Staubli VAL3: HRAS_trial.pjx

--- HRAS_trial.pjx ---
Parameters version=s7.10.2 stackSize=5000 millimeterUnit=true
Program file=calculate_pick.pgx
Program file=calculate_rc.pgx
Program file=calculate_total.pgx
Program file=check_out_set.pgx
Program file=f2_place.pgx
Program file=pick_cells.pgx
Program file=pp_auto_v1.pgx
Program file=pp_auto_v2.pgx
Program file=pp_bs_f1f2f3.pgx
Program file=pp_bs_f2f3.pgx
Program file=pp_cell_bk_f123.pgx
Program file=pp_cell_bk_f2f3.pgx
Program file=pp_cells.pgx
Program file=pp_shelf.pgx
Program file=regular_pick.pgx
Program file=regular_place.pgx
Program file=return_config.pgx
Program file=show_check.pgx
Program file=show_menu.pgx
Program file=show_progress.pgx
Program file=start.pgx
Program file=stop.pgx
Data file=HRAS_trial.dtx
Type name=vacuumSet path=Disk://designr0/designr0.pjx

--- HRAS_trial.dtx ---
dio dDio_t1_vb = {link=BasicIO-1\%Q1}
dio dDio_t1_vg
dio dDio_t1_vs = {link=fIn0}
dio dDio_t3_vb
dio dDio_t3_vg
dio dDio_t3_vs = {link=fIn0}
frame f1 = {x=-139.3, y=417.51507, z=-171.375326, rz=179.999983, fatherId=world[0]}
frame f2 = {x=-0.751213, y=410.035294, z=-169.439088, rz=179.999983, fatherId=world[0]}
frame f3 = {x=-105.214041, y=542.677355, z=-169.567493, rz=-89.997724, fatherId=world[0]}
frame fixture = {x=-479.290297, y=224.508367, z=-148, rz=-90.00005, fatherId=world[0]}
frame shelf = {x=-472.219676, y=345.637635, z=-165, rz=-90, fatherId=world[0]}
mdesc mNomSpeed
mdesc mSlowSpeed = {accel=50, vel=10, decel=50}
num nNum_blow_delay = 1
num nNum_blow_h = 0.5
num nNum_press = 4
num nNum_safe_h = 50
pointRx f1pick = {x=43.79, y=-7, z=0.5, rx=-180, rz=-180, fatherId=shelf[0]}
pointRx f1picksafe = {x=43.79, y=-7, z=20, rx=180, rz=-180, fatherId=shelf[0]}
pointRx f1place = {x=20, y=-19.98, rx=-180, rz=-180, fatherId=fixture[0]}
pointRx f1placesafe = {x=20, y=-19.98, z=20, rx=-180, rz=180, fatherId=fixture[0]}
pointRx f2pick = {x=29.79, y=-6.4, z=0.5, rx=-180, rz=180, fatherId=shelf[0]}
pointRx f2picksafe = {x=29.79, y=-6.4, z=20, rx=-180, rz=179, fatherId=shelf[0]}
pointRx f2place = {x=20, y=-16.82, rx=-180, rz=-180, fatherId=fixture[0]}
pointRx f2placesafe = {x=20, y=-16.82, z=20, rx=-180, rz=180, fatherId=fixture[0]}
pointRx f3pick = {x=7.79, y=-6.75, z=0.5, rx=-180, wrist=wpositive, fatherId=shelf[0]}
pointRx f3picksafe = {x=7.790741, y=-6.500263, z=50, rx=-179.999806, ry=-0.000248, rz=-2.000096, fatherId=shelf[0]}
pointRx f3place = {x=20, y=-16.62, z=3.8, rx=180, fatherId=fixture[0]}
pointRx f3placesafe = {x=20.000011, y=-16.619972, z=20, rx=-179.999664, ry=0.000116, rz=3E-06, fatherId=fixture[0]}
pointRx origin = {rx=-180, rz=-180, fatherId=fixture[0]}
pointRx pPointRx_f1_lb = {x=8.1, y=23.5, z=1.8, rx=180, fatherId=f1[0]}
pointRx pPointRx_f2_lb = {x=-3.5, y=25, z=0.2, rx=180, fatherId=f2[0]}
pointRx pPointRx_f3_lb = {x=28.5, y=3.34, z=0.2, rx=-180, rz=-180, fatherId=f3[0]}
pointRx ref = {x=-188.838954, y=475.816737, z=-162.486188, rx=180, rz=180, fatherId=world[0]}
screen sScreen_menu
screen sScreen_ppShelf
tool ca = {z=55, rz=45, fatherId=flange[0], ioLink=valve1}
tool t1 = {y=-18.5, fatherId=ca[0], ioLink=BasicIO-1\%Q0, ioOpen=1, ioClose=0.5}
tool t2 = {y=-4.5, fatherId=ca[0], ioLink=valve1}
tool t3 = {y=17.5, fatherId=ca[0], ioLink=BasicIO-1\%Q2, ioOpen=0.5, ioClose=0.5}
dio dDio_t1_cy
dio dDio_t2_cy
dio dDio_t3_cy

--- start.pgx ---
program start()
  local num l_nNum_choosen
begin
  resetMotion()

  //----------------------
  //  Reset I/O
  //----------------------
  call check_out_set(t1.gripper,false)
  call check_out_set(t2.gripper,false)
  call check_out_set(t3.gripper,false)

  call check_out_set(dDio_f1_fit,false)
  call check_out_set(dDio_bk,false)

  call check_out_set(dDio_f1_secure,false)
  call check_out_set(dDio_f2_secure,false)
  call check_out_set(dDio_f3_secure,false)

  call check_out_set(dDio_t1_cy,false)
  call check_out_set(dDio_t2_cy,false)
  call check_out_set(dDio_t3_cy,false)
  //----------------------
  //  Reset I/O
  //----------------------

  call show_menu(sScreen_ppShelf,l_nNum_choosen)

  while true
    switch l_nNum_choosen
      case 271
        //F1
        call pick_cells(1)
      break
      case 272
        //F2
        call pick_cells(2)
      break
      case 273
        //F3
        call pick_cells(3)
      break
      case 274
        //F4
        call pp_shelf()
      break
      case 275
        //F5
        call pp_cells()
      break
      //----------------------
      //
      //----------------------
      case 276
        //F6
        call pp_bs_f2f3()
      break
      case 277
        //F7
        call pp_auto_v1()
      break
      case 278
        //F8
        call pp_auto_v2()
      break
      case 113
        //q
        call pp_bs_f1f2f3()
      break
      default
        return
      break
    endSwitch
  endWhile

end

--- calculate_pick.pgx ---
public program calculate_pick(num x_nNum_row, num x_nNum_col, point& x_pPoint_return, num x_nNum_choose)
  local num l_nNum_pitchX
  local num l_nNum_pitchY
  local point l_pPoint_lb
begin
  //given row,col(z-based, count from left-bottom)
  //return position


  //set left-bottom corner position and pitch
  switch x_nNum_choose
    case 1
      //f1
      l_nNum_pitchX = 6.6
      l_nNum_pitchY = 11.3

      l_pPoint_lb = pPointRx_f1_lb
    break
    case 2
      //f2
      l_nNum_pitchX = 8
      l_nNum_pitchY = 10

      l_pPoint_lb = pPointRx_f2_lb
    break
    case 3
      //f3
      l_nNum_pitchX = -14
      l_nNum_pitchY = 22

      l_pPoint_lb = pPointRx_f3_lb
    break
    case 4
      //bottom
      l_nNum_pitchX = 32
      l_nNum_pitchY = 33

      l_pPoint_lb = pPointRx_bt_lb
    break

  endSwitch


  x_pPoint_return = l_pPoint_lb

  x_pPoint_return.trsf.x = x_pPoint_return.trsf.x + x_nNum_col * l_nNum_pitchX
  x_pPoint_return.trsf.y = x_pPoint_return.trsf.y + x_nNum_row * l_nNum_pitchY

  //---------------------------------------------
  // Bottom part special case - base frame offset
  //---------------------------------------------
  switch x_nNum_choose
    case 4
      fFrame_ofs.trsf.x = x_nNum_col * l_nNum_pitchX
      fFrame_ofs.trsf.y = x_nNum_row * l_nNum_pitchY
      //maintain the lb point
      x_pPoint_return = pPointRx_bt_lb
    break
  endSwitch

end

--- calculate_rc.pgx ---
program calculate_rc(num x_nNum_index, num x_nNum_choose, num& x_nNum_cRow, num& x_nNum_cCol)
  local num l_nNum_lCol
  local num l_nNum_lRow
begin

  call return_config(x_nNum_choose,l_nNum_lRow,l_nNum_lCol)

  //Quotien
  x_nNum_cRow = roundDown(x_nNum_index / (l_nNum_lCol + 1))
  //Modulo reminder
  x_nNum_cCol = x_nNum_index % (l_nNum_lCol+1)


end

--- calculate_total.pgx ---
program calculate_total(num x_nNum_choose, num& x_nNum_total)
  local num l_nNum_lCol
  local num l_nNum_lRow
begin
  call return_config(x_nNum_choose,l_nNum_lRow,l_nNum_lCol)
    //(max index)
  x_nNum_total = (l_nNum_lRow + 1) * (l_nNum_lCol+1)
end

--- check_out_set.pgx ---
program check_out_set(dio x_dDio_target, bool x_bBool_onoff)
begin
  if ioStatus(x_dDio_target) >= 0
    //once io is working
    x_dDio_target = x_bBool_onoff
  endIf
end

--- f1_cell_count.pgx ---
program f1_cell_count()
begin
  //given row,col , return position
  //retunr position
end

--- f1_cell_pick.pgx ---
program f1_cell_pick()
begin
  //pick from f1 put to bin
end

--- f2_place.pgx ---
program f2_place(mdesc x_mMdesc, mdesc x_mMdesc_slow)
  local point l_pPoint_blow
  local point l_pPoint_drop
  local point l_pPoint_safe
begin
  //vertical drop filter-2 process

  //control point preparation
  l_pPoint_safe=f2place
  l_pPoint_safe.trsf.z=l_pPoint_safe.trsf.z+nNum_safe_h

  l_pPoint_blow=f2place
  l_pPoint_blow.trsf.z=l_pPoint_blow.trsf.z+nNum_blow_h

  l_pPoint_drop=f2place

  ////to place via safe
  movej(l_pPoint_safe,t1,x_mMdesc)
  movej(l_pPoint_drop,t1,x_mMdesc)
  waitEndMove()
  //vg off
  if ioStatus(t1.gripper) >= 0
    close(t1)
  endIf
  if ioStatus(dDio_t1_vb) >= 0
    dDio_t1_vb=true
  endIf

    //on and delay
    delay(nNum_blow_delay)
    //to blow end
    movej(l_pPoint_blow,t1,x_mMdesc_slow)
    waitEndMove()
  //vb off
  if ioStatus(dDio_t1_vb) >= 0
     dDio_t1_vb=false
  endIf

    //to safe
    movej(l_pPoint_safe,t1,x_mMdesc)
    waitEndMove()
end

--- key_check.pgx ---
program key_check(string x_sString_show (dimensions=1))
begin
  userPage(sScreen_ppShelf)
  title(sScreen_ppShelf,x_sString_show)
  gotoxy(sScreen_ppShelf,0,6)
  putln(sScreen_ppShelf,"Press any key")
  //anykey
  get(sScreen_ppShelf)
  cls(sScreen_ppShelf)
end

--- pick_cells.pgx ---
program pick_cells(num x_nNum_choose)
  local num l_nNum_cRow
  local num l_nNum_cCol
  local point l_pPoint_cur
  local tool l_tTool_cur
  local point l_pPoint_lb_cur
  local num l_nNum_total
  local num l_nNum_current
  local dio l_dDio_cur_cy
  local dio l_dDio_secure
begin
  //pick from f1 put to bin
  call show_check("Reload")

  switch x_nNum_choose
    case 1
      //f1
      l_tTool_cur = t1
      dioLink(l_dDio_cur_cy,dDio_t1_cy)
      dioLink(l_dDio_secure,dDio_f1_secure)
      //dio assignment
    break
    case 2
      //f2
      l_tTool_cur = t2
      dioLink(l_dDio_cur_cy,dDio_t2_cy)
      dioLink(l_dDio_secure,dDio_f2_secure)
      //dio assignment
    break
    case 3
      //f3
      l_tTool_cur = t3
      dioLink(l_dDio_cur_cy,dDio_t3_cy)
      dioLink(l_dDio_secure,dDio_f3_secure)
      //dio assignment
    break

  endSwitch

  //calculate total
  call calculate_total(x_nNum_choose,l_nNum_total)

  for l_nNum_current=0 to(l_nNum_total-1) step 1

    //show progress
    call show_progress(sScreen_ppShelf,l_nNum_current+1,l_nNum_total,6)

    //row,col count
    call calculate_rc(l_nNum_current,x_nNum_choose,l_nNum_cRow,l_nNum_cCol)
    //pick position count
    call calculate_pick(l_nNum_cRow,l_nNum_cCol,l_pPoint_cur,x_nNum_choose)
    //pick (not defined yet
    call regular_pick(l_tTool_cur,mNomSpeed,mSlowSpeed,l_pPoint_cur,l_dDio_cur_cy,false,l_dDio_secure)

    //bin place (bin not defined yet
    call regular_place(l_tTool_cur,mNomSpeed,mSlowSpeed,ref,false,l_dDio_cur_cy,false)

  endFor

end

--- pickNplaceShelf.pgx ---
program pickNplaceShelf()
begin
  //assumption : arm in cal_ref1

  //pick f1
  //wait until user confirm (reload bottom
  //place f1
  //pick f2
  //wait until user confirm (close the fixture
  //place f2 (need blow simultanously
  //pick f3
  //place f3

end

--- place_f2.pgx ---
program place_f2()
begin
  //safe height
  //place
  //shut off
  dDio_t1_vg = off
  //back with blow

end

--- pp_auto_v1.pgx ---
program pp_auto_v1()
  local num l_nNum_bt_lim
  local num l_nNum_bt_idx
  local num l_nNum_f3_idx
  local num l_nNum_f2_idx
  local num l_nNum_f1_idx
  local num l_nNum_f3_lim
  local num l_nNum_f2_lim
  local num l_nNum_f1_lim
  local num l_nNum_cRow
  local num l_nNum_cCol
  local point l_pPoint_cur
begin
  //-----------------------------------------
  //  Cells to manual fixture
  //-----------------------------------------

  //initialize
  call calculate_total(1,l_nNum_f1_lim)
  call calculate_total(2,l_nNum_f2_lim)
  call calculate_total(3,l_nNum_f3_lim)
  call calculate_total(4,l_nNum_bt_lim)

  l_nNum_f1_idx = 0
  l_nNum_f2_idx = 0
  l_nNum_f3_idx = 0
  l_nNum_bt_idx = 0

  while true

    call show_check("Unload ASSY. filter")

    //------------
    //bottom cell pick
    //------------
    //runout remider
    if l_nNum_bt_idx >= l_nNum_bt_lim
      //warning if runs out
      call show_check("Reload Bottom")
      //reset
      l_nNum_bt_idx = 0
    endIf


    call calculate_rc(l_nNum_bt_idx,4,l_nNum_cRow,l_nNum_cCol)
    call calculate_pick(l_nNum_cRow,l_nNum_cCol,l_pPoint_cur,4)
    call regular_pick(t3,mNomSpeed,mSlowSpeed,l_pPoint_cur,dDio_t3_cy,false,dDio_f3_secure)

    //show progress
    call show_progress(sScreen_ppShelf,l_nNum_bt_idx+1,l_nNum_bt_lim,5)
    //increase
    l_nNum_bt_idx = l_nNum_bt_idx +1

    //------------
    //bottom place
    //------------
    call regular_place(t3,mNomSpeed,mSlowSpeed,pPointRx_bt_pos,false,dDio_t3_cy,false)

    //------------
    //f1 cell pick
    //------------

    //runout remider
    if l_nNum_f1_idx >= l_nNum_f1_lim
      //warning if runs out
      call show_check("Reload F1")
      //reset
      l_nNum_f1_idx = 0
    endIf

    call calculate_rc(l_nNum_f1_idx,1,l_nNum_cRow,l_nNum_cCol)
    call calculate_pick(l_nNum_cRow,l_nNum_cCol,l_pPoint_cur,1)
    call regular_pick(t1,mNomSpeed,mSlowSpeed,l_pPoint_cur,dDio_t1_cy,false,dDio_f1_secure)

    //show progress
    call show_progress(sScreen_ppShelf,l_nNum_f1_idx+1,l_nNum_f1_lim,6)
    //increase
    l_nNum_f1_idx = l_nNum_f1_idx +1

    //----------
    //f2 cell pick
    //------------

    //runout remider
    if l_nNum_f2_idx >= l_nNum_f2_lim
      //warning if runs out
      call show_check("Reload F2")
      //reset
      l_nNum_f2_idx = 0
    endIf


    call calculate_rc(l_nNum_f2_idx,2,l_nNum_cRow,l_nNum_cCol)
    call calculate_pick(l_nNum_cRow,l_nNum_cCol,l_pPoint_cur,2)
    call regular_pick(t2,mNomSpeed,mSlowSpeed,l_pPoint_cur,dDio_t2_cy,false,dDio_f2_secure)
    //show progress
    call show_progress(sScreen_ppShelf,l_nNum_f2_idx+1,l_nNum_f2_lim,7)
    //increase
    l_nNum_f2_idx = l_nNum_f2_idx +1

    //-------
    //f3pick
    //-------

    //runout reminder
    if l_nNum_f3_idx >= l_nNum_f3_lim
      //warning if runs out
      call show_check("Reload F3")
      //reset
      l_nNum_f3_idx = 0
    endIf
    call calculate_rc(l_nNum_f3_idx,3,l_nNum_cRow,l_nNum_cCol)
    call calculate_pick(l_nNum_cRow,l_nNum_cCol,l_pPoint_cur,3)
    call regular_pick(t3,mNomSpeed,mSlowSpeed,l_pPoint_cur,dDio_t3_cy,false,dDio_f3_secure)

    //show progress
    call show_progress(sScreen_ppShelf,l_nNum_f3_idx+1,l_nNum_f3_lim,8)
    //increase
    l_nNum_f3_idx = l_nNum_f3_idx +1

    //-------------
    // Back secure
    //-------------
    call pp_bs_f2f3()

    //----------------
    // F1, F2+F3 place
    //----------------
    call regular_place(t1,mNomSpeed,mSlowSpeed,pPointRx_f1_pos,false,dDio_t1_cy,false)
    // put  f1 fit
    if ioStatus(dDio_f1_fit) >= 0
      dDio_f1_fit = true
      delay(nNum_cy_delay)
    endIf
    //f3place
    call regular_place(t3,mNomSpeed,mSlowSpeed,pPointRx_f3_pos,false,dDio_t3_cy,false)
    // off  f1 fit
    if ioStatus(dDio_f1_fit) >= 0
      dDio_f1_fit = false
    endIf

  endWhile


end

--- pp_auto_v2.pgx ---
program pp_auto_v2(bool x_bBool_single)
  local num l_nNum_bt_lim
  local num l_nNum_bt_idx
  local num l_nNum_f3_idx
  local num l_nNum_f2_idx
  local num l_nNum_f1_idx
  local num l_nNum_f3_lim
  local num l_nNum_f2_lim
  local num l_nNum_f1_lim
  local num l_nNum_cRow
  local num l_nNum_cCol
  local point l_pPoint_cur
begin
  //-----------------------------------------
  //  Cells to manual fixture
  //-----------------------------------------

  //initialize
  call calculate_total(1,l_nNum_f1_lim)
  call calculate_total(2,l_nNum_f2_lim)
  call calculate_total(3,l_nNum_f3_lim)
  call calculate_total(4,l_nNum_bt_lim)

  l_nNum_f1_idx = 0
  l_nNum_f2_idx = 0
  l_nNum_f3_idx = 0
  l_nNum_bt_idx = 0

  while true

    call show_check("Unload ASSY. filter")

    if x_bBool_single == true
      //prompt reminder
      l_nNum_bt_idx = l_nNum_bt_lim
    endIf

    //------------
    //bottom cell pick
    //------------
    //runout remider
    if l_nNum_bt_idx >= l_nNum_bt_lim
      //warning if runs out
      call show_check("Reload Bottom")
      //reset
      l_nNum_bt_idx = 0
    endIf

    call calculate_rc(l_nNum_bt_idx,4,l_nNum_cRow,l_nNum_cCol)
    call calculate_pick(l_nNum_cRow,l_nNum_cCol,l_pPoint_cur,4)
    call regular_pick(t3,mNomSpeed,mSlowSpeed,l_pPoint_cur,dDio_t3_cy,false,dDio_f3_secure)


    //show progress
    call show_progress(sScreen_ppShelf,l_nNum_bt_idx+1,l_nNum_bt_lim,5)
    //increase
    l_nNum_bt_idx = l_nNum_bt_idx +1

    //------------
    //bottom place
    //------------
    call regular_place(t3,mNomSpeed,mSlowSpeed,pPointRx_bt_pos,false,dDio_t3_cy,false)

    //------------
    //f1 cell pick
    //------------

    //runout remider
    if l_nNum_f1_idx >= l_nNum_f1_lim
      //warning if runs out
      call show_check("Reload F1")
      //reset
      l_nNum_f1_idx = 0
    endIf

    call calculate_rc(l_nNum_f1_idx,1,l_nNum_cRow,l_nNum_cCol)
    call calculate_pick(l_nNum_cRow,l_nNum_cCol,l_pPoint_cur,1)
    call regular_pick(t1,mNomSpeed,mSlowSpeed,l_pPoint_cur,dDio_t1_cy,false,dDio_f1_secure)

    //show progress
    call show_progress(sScreen_ppShelf,l_nNum_f1_idx+1,l_nNum_f1_lim,6)
    //increase
    l_nNum_f1_idx = l_nNum_f1_idx +1

    //----------
    //f2 cell pick
    //------------

    //runout remider
    if l_nNum_f2_idx >= l_nNum_f2_lim
      //warning if runs out
      call show_check("Reload F2")
      //reset
      l_nNum_f2_idx = 0
    endIf


    call calculate_rc(l_nNum_f2_idx,2,l_nNum_cRow,l_nNum_cCol)
    call calculate_pick(l_nNum_cRow,l_nNum_cCol,l_pPoint_cur,2)
    call regular_pick(t2,mNomSpeed,mSlowSpeed,l_pPoint_cur,dDio_t2_cy,false,dDio_f2_secure)
    //show progress
    call show_progress(sScreen_ppShelf,l_nNum_f2_idx+1,l_nNum_f2_lim,7)
    //increase
    l_nNum_f2_idx = l_nNum_f2_idx +1

    //-------
    //f3pick
    //-------

    //runout reminder
    if l_nNum_f3_idx >= l_nNum_f3_lim
      //warning if runs out
      call show_check("Reload F3")
      //reset
      l_nNum_f3_idx = 0
    endIf
    call calculate_rc(l_nNum_f3_idx,3,l_nNum_cRow,l_nNum_cCol)
    call calculate_pick(l_nNum_cRow,l_nNum_cCol,l_pPoint_cur,3)
    call regular_pick(t3,mNomSpeed,mSlowSpeed,l_pPoint_cur,dDio_t3_cy,false,dDio_f3_secure)

    //show progress
    call show_progress(sScreen_ppShelf,l_nNum_f3_idx+1,l_nNum_f3_lim,8)
    //increase
    l_nNum_f3_idx = l_nNum_f3_idx +1

    //-------------
    // Back secure (F1,F2,F3
    //-------------
    call pp_bs_f1f2f3()
    //-------------
    // F1,F2,F3 pick at once
    //-------------
    call regular_pick(t3,mNomSpeed,mSlowSpeed,pPointRx_f3_bk,dDio_t3_cy,false,dDio_f3_secure)
    //----------------
    // F1+F2+F3 place at once
    //----------------
    //f3place
    call regular_place(t3,mNomSpeed,mSlowSpeed,pPointRx_f3_pos,false,dDio_t3_cy,false)

  endWhile


end

--- pp_back_secure.pgx ---
program pp_back_secure()
begin
  //given f2,f3 are in hand
  //exit state : f2, f3 secured in one hand

  //place f2 in origin of bk (//open bk vacuum
  call regular_place(t2,mNomSpeed,mSlowSpeed,pPointRx_f2_bk,false,dDio_t2_cy,true)

  //drop f3 offset from f2 origin
  call regular_pick(t3,mNomSpeed,mSlowSpeed,pPointRx_f3_bk,dDio_t3_cy,false,dDio_f3_secure)

end

--- pp_bs_f1f2f3.pgx ---
program pp_bs_f1f2f3()
begin
  //given f1,f2,f3 are in hand
  //exit state : f1,f2,f3 secured in bs

  //place f2 in origin of bk (//open bk vacuum
  call regular_place(t1,mNomSpeed,mSlowSpeed,pPointRx_f1_bk,false,dDio_t1_cy,true)

  //place f2 in origin of bk (//open bk vacuum
  call regular_place(t2,mNomSpeed,mSlowSpeed,pPointRx_f2_bk,false,dDio_t2_cy,true)

  //drop f3 offset from f2 origin
  call regular_place(t3,mNomSpeed,mSlowSpeed,pPointRx_f3_bk,false,dDio_t3_cy,true)

end

--- pp_bs_f2f3.pgx ---
program pp_bs_f2f3()
begin
  //given f2,f3 are in hand
  //exit state : f2, f3 secured in one hand

  //place f2 in origin of bk (//open bk vacuum
  call regular_place(t2,mNomSpeed,mSlowSpeed,pPointRx_f2_bk,false,dDio_t2_cy,true)

  //drop f3 offset from f2 origin
  call regular_pick(t3,mNomSpeed,mSlowSpeed,pPointRx_f3_bk,dDio_t3_cy,false,dDio_f3_secure)

end

--- pp_cell_bk.pgx ---
program pp_cell_bk()
  local num l_nNum_f2_lim
  local num l_nNum_f3_lim
  local num l_nNum_f2_idx
  local num l_nNum_f3_idx
  local num l_nNum_cRow
  local num l_nNum_cCol
  local point l_pPoint_cur
begin
  //---------------------------------
  //from cells(f2,f3) to back secure
  //---------------------------------

   //initialize
  call calculate_total(2,l_nNum_f2_lim)
  call calculate_total(3,l_nNum_f3_lim)

  l_nNum_f2_idx = 0
  l_nNum_f3_idx = 0

  while true

    //reload  reminder
    call show_check("Recycle pp_cell_bk")

    //----------
    //f2 cell pick
    //------------

    //runout remider
    if l_nNum_f2_idx >= l_nNum_f2_lim
      //warning if runs out
      call show_check("Reload F2")
      //reset
      l_nNum_f2_idx = 0
    endIf

    call calculate_rc(l_nNum_f2_idx,2,l_nNum_cRow,l_nNum_cCol)
    call calculate_pick(l_nNum_cRow,l_nNum_cCol,l_pPoint_cur,2)
    call regular_pick(t2,mNomSpeed,mSlowSpeed,l_pPoint_cur,dDio_t2_cy,false,dDio_f2_secure)
    //show progress
    call show_progress(sScreen_ppShelf,l_nNum_f2_idx+1,l_nNum_f2_lim,7)
    //increase
    l_nNum_f2_idx = l_nNum_f2_idx +1

    //-------
    //f3pick
    //-------

    //runout reminder
    if l_nNum_f3_idx >= l_nNum_f3_lim
      //warning if runs out
      call show_check("Reload F3")
      //reset
      l_nNum_f3_idx = 0
    endIf
    call calculate_rc(l_nNum_f3_idx,3,l_nNum_cRow,l_nNum_cCol)
    call calculate_pick(l_nNum_cRow,l_nNum_cCol,l_pPoint_cur,3)
    call regular_pick(t3,mNomSpeed,mSlowSpeed,l_pPoint_cur,dDio_t3_cy,false,dDio_f3_secure)
    //show progress
    call show_progress(sScreen_ppShelf,l_nNum_f3_idx+1,l_nNum_f3_lim,8)
    //increase
    l_nNum_f3_idx = l_nNum_f3_idx +1

    //--------------
    //pp back secure
    //--------------
    call pp_back_secure()

    //-------------
    // drop
    //-------------
    call regular_place(t3,mNomSpeed,mSlowSpeed,pPointRx_f3_bk,false,dDio_t3_cy,false)


  endWhile


end

--- pp_cell_bk_f123.pgx ---
program pp_cell_bk_f123()
  local num l_nNum_f1_idx
  local num l_nNum_f1_lim
  local num l_nNum_f2_lim
  local num l_nNum_f3_lim
  local num l_nNum_f2_idx
  local num l_nNum_f3_idx
  local num l_nNum_cRow
  local num l_nNum_cCol
  local point l_pPoint_cur
begin
  //---------------------------------
  //from cells(f1,f2,f3) to back secure
  //---------------------------------

  //initialize
  call calculate_total(1,l_nNum_f1_lim)
  call calculate_total(2,l_nNum_f2_lim)
  call calculate_total(3,l_nNum_f3_lim)

  l_nNum_f1_idx = 0
  l_nNum_f2_idx = 0
  l_nNum_f3_idx = 0

  while true

    //reload  reminder
    call show_check("Recycle pp_cell_bk")

    //------------
    //f1 cell pick
    //------------

    //runout remider
    if l_nNum_f1_idx >= l_nNum_f1_lim
      //warning if runs out
      call show_check("Reload F1")
      //reset
      l_nNum_f1_idx = 0
    endIf

    call calculate_rc(l_nNum_f1_idx,1,l_nNum_cRow,l_nNum_cCol)
    call calculate_pick(l_nNum_cRow,l_nNum_cCol,l_pPoint_cur,1)
    call regular_pick(t1,mNomSpeed,mSlowSpeed,l_pPoint_cur,dDio_t1_cy,false,dDio_f1_secure)

    //show progress
    call show_progress(sScreen_ppShelf,l_nNum_f1_idx+1,l_nNum_f1_lim,6)
    //increase
    l_nNum_f1_idx = l_nNum_f1_idx +1

    //----------
    //f2 cell pick
    //------------

    //runout remider
    if l_nNum_f2_idx >= l_nNum_f2_lim
      //warning if runs out
      call show_check("Reload F2")
      //reset
      l_nNum_f2_idx = 0
    endIf

    call calculate_rc(l_nNum_f2_idx,2,l_nNum_cRow,l_nNum_cCol)
    call calculate_pick(l_nNum_cRow,l_nNum_cCol,l_pPoint_cur,2)
    call regular_pick(t2,mNomSpeed,mSlowSpeed,l_pPoint_cur,dDio_t2_cy,false,dDio_f2_secure)
    //show progress
    call show_progress(sScreen_ppShelf,l_nNum_f2_idx+1,l_nNum_f2_lim,7)
    //increase
    l_nNum_f2_idx = l_nNum_f2_idx +1

    //-------
    //f3pick
    //-------

    //runout reminder
    if l_nNum_f3_idx >= l_nNum_f3_lim
      //warning if runs out
      call show_check("Reload F3")
      //reset
      l_nNum_f3_idx = 0
    endIf
    call calculate_rc(l_nNum_f3_idx,3,l_nNum_cRow,l_nNum_cCol)
    call calculate_pick(l_nNum_cRow,l_nNum_cCol,l_pPoint_cur,3)
    call regular_pick(t3,mNomSpeed,mSlowSpeed,l_pPoint_cur,dDio_t3_cy,false,dDio_f3_secure)
    //show progress
    call show_progress(sScreen_ppShelf,l_nNum_f3_idx+1,l_nNum_f3_lim,8)
    //increase
    l_nNum_f3_idx = l_nNum_f3_idx +1

    //--------------
    //pp back secure
    //--------------
    call pp_bs_f1f2f3()

  endWhile


end

--- pp_cell_bk_f2f3.pgx ---
program pp_cell_bk_f2f3()
  local num l_nNum_f2_lim
  local num l_nNum_f3_lim
  local num l_nNum_f2_idx
  local num l_nNum_f3_idx
  local num l_nNum_cRow
  local num l_nNum_cCol
  local point l_pPoint_cur
begin
  //---------------------------------
  //from cells(f2,f3) to back secure
  //---------------------------------

   //initialize
  call calculate_total(2,l_nNum_f2_lim)
  call calculate_total(3,l_nNum_f3_lim)

  l_nNum_f2_idx = 0
  l_nNum_f3_idx = 0

  while true

    //reload  reminder
    call show_check("Recycle pp_cell_bk")

    //----------
    //f2 cell pick
    //------------

    //runout remider
    if l_nNum_f2_idx >= l_nNum_f2_lim
      //warning if runs out
      call show_check("Reload F2")
      //reset
      l_nNum_f2_idx = 0
    endIf

    call calculate_rc(l_nNum_f2_idx,2,l_nNum_cRow,l_nNum_cCol)
    call calculate_pick(l_nNum_cRow,l_nNum_cCol,l_pPoint_cur,2)
    call regular_pick(t2,mNomSpeed,mSlowSpeed,l_pPoint_cur,dDio_t2_cy,false,dDio_f2_secure)
    //show progress
    call show_progress(sScreen_ppShelf,l_nNum_f2_idx+1,l_nNum_f2_lim,7)
    //increase
    l_nNum_f2_idx = l_nNum_f2_idx +1

    //-------
    //f3pick
    //-------

    //runout reminder
    if l_nNum_f3_idx >= l_nNum_f3_lim
      //warning if runs out
      call show_check("Reload F3")
      //reset
      l_nNum_f3_idx = 0
    endIf
    call calculate_rc(l_nNum_f3_idx,3,l_nNum_cRow,l_nNum_cCol)
    call calculate_pick(l_nNum_cRow,l_nNum_cCol,l_pPoint_cur,3)
    call regular_pick(t3,mNomSpeed,mSlowSpeed,l_pPoint_cur,dDio_t3_cy,false,dDio_f3_secure)
    //show progress
    call show_progress(sScreen_ppShelf,l_nNum_f3_idx+1,l_nNum_f3_lim,8)
    //increase
    l_nNum_f3_idx = l_nNum_f3_idx +1

    //--------------
    //pp back secure
    //--------------
    call pp_bs_f2f3()

    //-------------
    // drop
    //-------------
    call regular_place(t3,mNomSpeed,mSlowSpeed,pPointRx_f3_bk,false,dDio_t3_cy,false)


  endWhile


end

--- pp_cells.pgx ---
program pp_cells()
  local num l_nNum_f3_idx
  local num l_nNum_f2_idx
  local num l_nNum_f1_idx
  local num l_nNum_f3_lim
  local num l_nNum_f2_lim
  local num l_nNum_f1_lim
  local num l_nNum_cRow
  local num l_nNum_cCol
  local point l_pPoint_cur
begin
  //-----------------------------------------
  //  Cells to manual fixture
  //-----------------------------------------

  //initialize
  call calculate_total(1,l_nNum_f1_lim)
  call calculate_total(2,l_nNum_f2_lim)
  call calculate_total(3,l_nNum_f3_lim)

  l_nNum_f1_idx = 0
  l_nNum_f2_idx = 0
  l_nNum_f3_idx = 0

  while true
    //reload bottom reminder
    call show_check("Reload bottom")

    //------------
    //f1 cell pick
    //------------

    //runout remider
    if l_nNum_f1_idx >= l_nNum_f1_lim
      //warning if runs out
      call show_check("Reload F1")
      //reset
      l_nNum_f1_idx = 0
    endIf


    call calculate_rc(l_nNum_f1_idx,1,l_nNum_cRow,l_nNum_cCol)
    call calculate_pick(l_nNum_cRow,l_nNum_cCol,l_pPoint_cur,1)

    call regular_pick(t1,mNomSpeed,mSlowSpeed,l_pPoint_cur,dDio_t1_cy,false,dDio_f1_secure)
    //f1 place
    call regular_place(t1,mNomSpeed,mSlowSpeed,f1place,false,dDio_t1_cy,false)

    //show progress
    call show_progress(sScreen_ppShelf,l_nNum_f1_idx+1,l_nNum_f1_lim,6)
    //increase
    l_nNum_f1_idx = l_nNum_f1_idx +1


    //----------
    //f2 cell pick
    //------------

    //runout remider
    if l_nNum_f2_idx >= l_nNum_f2_lim
      //warning if runs out
      call show_check("Reload F2")
      //reset
      l_nNum_f2_idx = 0
    endIf


    call calculate_rc(l_nNum_f2_idx,2,l_nNum_cRow,l_nNum_cCol)
    call calculate_pick(l_nNum_cRow,l_nNum_cCol,l_pPoint_cur,2)
    call regular_pick(t2,mNomSpeed,mSlowSpeed,l_pPoint_cur,dDio_t2_cy,false,dDio_f2_secure)
    //fixture reminder
    call show_check("Place fixture")
    //f2 place
    call f2_place(mNomSpeed,mSlowSpeed)

    //show progress
    call show_progress(sScreen_ppShelf,l_nNum_f2_idx+1,l_nNum_f2_lim,7)
    //increase
    l_nNum_f2_idx = l_nNum_f2_idx +1

    //-------
    //f3pick
    //-------

    //runout reminder
    if l_nNum_f3_idx >= l_nNum_f3_lim
      //warning if runs out
      call show_check("Reload F3")
      //reset
      l_nNum_f3_idx = 0
    endIf
    call calculate_rc(l_nNum_f3_idx,3,l_nNum_cRow,l_nNum_cCol)
    call calculate_pick(l_nNum_cRow,l_nNum_cCol,l_pPoint_cur,3)

    call regular_pick(t3,mNomSpeed,mSlowSpeed,l_pPoint_cur,dDio_t3_cy,false,dDio_f3_secure)
    //f3place
    call regular_place(t3,mNomSpeed,mSlowSpeed,f3place,true,dDio_t3_cy,false)

    //show progress
    call show_progress(sScreen_ppShelf,l_nNum_f3_idx+1,l_nNum_f3_lim,8)
    //increase
    l_nNum_f3_idx = l_nNum_f3_idx +1

  endWhile


end

--- pp_shelf.pgx ---
program pp_shelf()
begin
  //pick and place procedure shelf-fixture
  //assumed that start from cal_ref_1

  //show message and get input (if reloaded all material
  call show_check("Reload")

  //f1 pick and palce
  call regular_pick(t1,mNomSpeed,mSlowSpeed,f1pick,dDio_t1_cy,false,dDio_f1_secure)
  call regular_place(t1,mNomSpeed,mSlowSpeed,f1place,false,dDio_t1_cy,false)

  //f2 pick and place
  call regular_pick(t1,mNomSpeed,mSlowSpeed,f2pick,dDio_t1_cy,false,dDio_f1_secure)
  //show message and get input (if fixture applied
  call show_check("Fixture close")

  call f2_place(mNomSpeed,mSlowSpeed)

  //f3 pick and place
  call regular_pick(t3,mNomSpeed,mSlowSpeed,f3pick,dDio_t3_cy,false,dDio_f3_secure)
  call regular_place(t3,mNomSpeed,mSlowSpeed,f3place,true,dDio_t3_cy,false)

end

--- regular_pick.pgx ---
program regular_pick(tool x_tTool, mdesc x_mMdesc, mdesc x_mMdesc_slow, point x_pPoint_pick, dio x_dDio_cy, bool x_bBool_bk, dio x_dDio_secure)
  local point l_pPoint_pick
  local point l_pPoint_safe
  local point l_pPoint_aprch
begin

  //vertical regular pick process

  //control point preparation
  l_pPoint_safe=x_pPoint_pick
  l_pPoint_safe.trsf.z=l_pPoint_safe.trsf.z+nNum_safe_h
  //approach point preparation
  l_pPoint_aprch=x_pPoint_pick
  l_pPoint_aprch.trsf.z=l_pPoint_aprch.trsf.z+nNum_apporach_h
  //pick point preparation
  l_pPoint_pick=x_pPoint_pick

  ////to place via safe (in sequence)
  movej(l_pPoint_safe,x_tTool,x_mMdesc)
  waitEndMove()

  //corresponding cylinder extend
  if ioStatus(x_dDio_cy) >= 0
    //once io is working , on
    x_dDio_cy = true
    delay(nNum_cy_delay)
  endIf

  //open secure (on the cell not on the back secure
  if !x_bBool_bk
    call check_out_set(x_dDio_secure,true)
  endIf

  //---------------------------------
  // vertical should be linear mode
  // (Fast approach
  //---------------------------------
  movel(l_pPoint_aprch,x_tTool,x_mMdesc)
  waitEndMove()
  //---------------------------------
  // vertical should be linear mode
  // (Slow pick
  //---------------------------------
  movel(l_pPoint_pick,x_tTool,x_mMdesc_slow)
  waitEndMove()

  //vg on
  if ioStatus(x_tTool.gripper) >= 0
    //once io is working
    open(x_tTool)
  endIf

  //activate/deactive back secure if any
  if ioStatus(dDio_bk) >= 0
    //once dDio_bk is working
    dDio_bk = x_bBool_bk
    //delay to release
    delay(nNum_blow_delay)
  endIf

  //----------
  //to safe
  // (Slow up
  //----------
  movel(l_pPoint_aprch,x_tTool,x_mMdesc_slow)
  waitEndMove()
  //----------
  //to safe
  // (Fast
  //----------
  movel(l_pPoint_safe,x_tTool,x_mMdesc)
  waitEndMove()

  //corresponding cylinder extract
  if ioStatus(x_dDio_cy) >= 0
    //once io is working , off
    x_dDio_cy = false
  endIf

  //shut secure
  call check_out_set(x_dDio_secure,false)

  //check if vacuum established
  //if x_bBool_check and (dioGet(x_dDio_vs)==1)
  //success
  //elseIf x_bBool_check and (dioGet(x_dDio_vs)==1)
  //failed
  //else
  //irrelevant from IO check
  //endIf

end

--- regular_place.pgx ---
program regular_place(tool x_tTool, mdesc x_mMdesc, mdesc x_mMdesc_slow, point x_pPoint_place, bool x_bBool_press, dio x_dDio_cy, bool x_bBool_bk)
  local point l_pPoint_drop
  local point l_pPoint_safe
  local point l_pPoint_press
  local point l_pPoint_aprch
begin
  //vertical regular drop process

  //----------------------------
  //control point preparation
  //----------------------------
  l_pPoint_safe=x_pPoint_place
  l_pPoint_safe.trsf.z=l_pPoint_safe.trsf.z+nNum_safe_h
  //----------------------------
  //approach point preparation
  //----------------------------
  l_pPoint_aprch=x_pPoint_place
  l_pPoint_aprch.trsf.z=l_pPoint_aprch.trsf.z+nNum_apporach_h
  //----------------------------
  //place point preparation
  //----------------------------
  l_pPoint_drop=x_pPoint_place

  l_pPoint_press = x_pPoint_place
  l_pPoint_press.trsf.z = l_pPoint_press.trsf.z-nNum_press

  ////to place via safe
  movej(l_pPoint_safe,x_tTool,x_mMdesc)
  waitEndMove()

  //corresponding cylinder extend
  if ioStatus(x_dDio_cy) >= 0
    //once io is working , on
    x_dDio_cy = true
    delay(nNum_cy_delay)
  endIf

  //---------------------------------
  // vertical should be linear mode
  // (Fast approach
  //---------------------------------
  movel(l_pPoint_aprch,x_tTool,x_mMdesc)
  waitEndMove()
  //---------------------------------
  // vertical should be linear mode
  //---------------------------------
  movel(l_pPoint_drop,x_tTool,x_mMdesc_slow)
  waitEndMove()
  //vg off
  if ioStatus(x_tTool.gripper) >= 0
    //once io is working
    close(x_tTool)
  endIf

  //additional press
  if x_bBool_press
    //---------------------------------
    // vertical should be linear mode
    //---------------------------------
    movel(l_pPoint_press,x_tTool,x_mMdesc)
    waitEndMove()
  endIf

  //additional back secure
  if ioStatus(dDio_bk) >= 0
    //once io is working and require back secure, on
    dDio_bk = x_bBool_bk
  endIf

  //----------
  //to safe
  // (Slow up
  //----------
  movel(l_pPoint_aprch,x_tTool,x_mMdesc_slow)
  waitEndMove()
  //---------------------------------
  // vertical should be linear mode
  //---------------------------------
  //to safe
  movel(l_pPoint_safe,x_tTool,x_mMdesc)
  waitEndMove()

  //corresponding cylinder extract
  if ioStatus(x_dDio_cy) >= 0
    //once io is working , off
    x_dDio_cy = false
  endIf

end

--- return_config.pgx ---
program return_config(num x_nNum_choose, num& x_nNum_lRow, num& x_nNum_lCol)
begin

   switch x_nNum_choose
    case 1
      //f1
      x_nNum_lCol = 5
      x_nNum_lRow = 5
    break
    case 2
      //f2
      x_nNum_lCol = 11
      x_nNum_lRow = 2
    break
    case 3
      //f3
      //x_nNum_lCol = 2
      //x_nNum_lRow = 5

      x_nNum_lCol = 5
      x_nNum_lRow = 2
    break
    case 4
      //bottom
      x_nNum_lCol = 2
      x_nNum_lRow = 5
    break

  endSwitch

end

--- show_check.pgx ---
program show_check(string x_sString_show)
begin
  userPage(sScreen_ppShelf)
  title(sScreen_ppShelf,x_sString_show)
  gotoxy(sScreen_ppShelf,0,0)
  putln(sScreen_ppShelf,"Press any key")
  //anykey
  get(sScreen_ppShelf)
  //cls(sScreen_ppShelf)
end

--- show_menu.pgx ---
program show_menu(screen& x_sScreen, num& x_nNum_choosed)
begin


  userPage(x_sScreen)
  title(x_sScreen,"Choose sub")

  gotoxy(x_sScreen,0,0)
  putln(x_sScreen,"F1)Filter 1 pick/bin")
  gotoxy(x_sScreen,0,1)
  putln(x_sScreen,"F2)Filter 2 pick/bin")
  gotoxy(x_sScreen,0,2)
  putln(x_sScreen,"F3)Filter 3 pick/bin")
  gotoxy(x_sScreen,0,3)
  putln(x_sScreen,"F4)Shelf pick/fixture (depreciated)")
  gotoxy(x_sScreen,0,4)
  putln(x_sScreen,"F5)Assemble")
  //---------------
  //  HRAS Lite
  //---------------
  gotoxy(x_sScreen,0,5)
  putln(x_sScreen,"F6)Cell to back secure f2f3")
  gotoxy(x_sScreen,0,6)
  putln(x_sScreen,"F7)Auto ver1")
  gotoxy(x_sScreen,0,7)
  putln(x_sScreen,"F8)Auto ver2")
  gotoxy(x_sScreen,0,8)
  putln(x_sScreen,"q)Cell to back secure f1f2f3")

  //anykey
  x_nNum_choosed = get(x_sScreen)
  cls(x_sScreen)
end

--- show_progress.pgx ---
program show_progress(screen& x_sScreen, num x_nNum_run, num x_nNum_total, num x_nNum_row)
begin
    userPage(sScreen_ppShelf)
  title(sScreen_ppShelf,"Progree")
  gotoxy(sScreen_ppShelf,0,x_nNum_row)

  putln(sScreen_ppShelf, toString("",x_nNum_run) + "/" + toString("",x_nNum_total))
end
